{attribute addProperty BoxType "EL1258-0000-0016"}
{attribute addProperty Id "StatusAT %I*Status_8577222D607.51InputsAT %I*Inputs_8B7B380018623.2533Input_event_timeAT %I*ARRAY[0 ..9] OF UDINT320400"}
{attribute addProperty CRC "3582494864"}
{attribute addProperty SizeInBites "566"}
{attribute addProperty SizeInBytes "70.75"}
TYPE MTI_Inputs_10x_Channel_D2104A60 :
STRUCT
	{attribute addProperty Name "Status"}
	Status AT %I* : Status_8577222D;
	{attribute addProperty Name "Inputs"}
	Inputs AT %I* : Inputs_8B7B3800;
	{attribute addProperty Name "Input_event_time"}
	Input_event_time AT %I* : ARRAY[0 ..9] OF UDINT;
END_STRUCT
END_TYPE

(* stored: Version 1.2.0.0, ProductVersion 3.1.4024.9
   DUT MTI_Inputs_10x_Channel_D2104A60: Id {af918b00-05a4-40d6-a1e0-6e92829772cc} *)
